Fanuc KAREL source: kx00011.KL

-- PROVISIONAL review KL for V1013-1; original PC SHA256 ee63c9b85606f4b063b1c19fee645adfd44953bb0b58ef3ba6b5889dcbd51cc6
-- Incomplete behavior may be omitted. Consult companion uncertainty JSON. Do not deploy.
PROGRAM KX00011
%NOLOCKGROUP
VAR
  I : INTEGER
  J : INTEGER
  B : BOOLEAN
  F : FILE
  S : STRING[80]
-- UNRESOLVED_DECL P type=000102
BEGIN
  -- UNRESOLVED_PC offsets 5-7; opcodes 9C,65
  -- UNRESOLVED_PC offsets 12-16; opcodes 7F
END KX00011
